(* CoDeSys 2.3 export: geometry.st *)

(* POU Math/Geometry/CIRCLE_A, ST *)
FUNCTION CIRCLE_A : REAL
VAR_INPUT
	R : REAL;
END_VAR


(*
version 1.1	18. oct. 2008
programmer 	hugo
tested by	oscat

this function calculates the area of a circle with radius R

*)
CIRCLE_A := R * R * math.PI;


(* revision history
hm	22. jan. 2007	rev 1.0
	original version

hm	18. oct. 2008	rev 1.1
	using math constants

*)
END_FUNCTION

(* POU Math/Geometry/CIRCLE_C, ST *)
FUNCTION CIRCLE_C : REAL
VAR_INPUT
	R : REAL;
END_VAR


(*
version 1.1	18. oct. 2008
programmer 	hugo
tested by	oscat

this function calculates the circumference of a circle with radius R

*)
CIRCLE_C := R * math.PI2;


(* revision history
hm	22. jan. 2007	rev 1.0
	original version

hm	18. oct. 2008	rev 1.1
	using math constants

*)
END_FUNCTION

(* POU Math/Geometry/CIRCLE_SEG, ST *)
FUNCTION CIRCLE_SEG : REAL
VAR_INPUT
	R : REAL;
	A : REAL;
END_VAR


(*
version 1.1	18. oct. 2008
programmer 	hugo
tested by	oscat

this function calculates the area of a circle segment with radius R and angle A

*)
CIRCLE_SEG := R * R * math.PI * A / 360.0;


(* revision history
hm	22. jan. 2007	rev 1.0
	original version

hm	18. oct. 2008	rev 1.1
	using math constants

*)
END_FUNCTION

(* POU Math/Geometry/CONE_V, ST *)
FUNCTION CONE_V : REAL
VAR_INPUT
	R : REAL;
	H : REAL;
END_VAR


(*
version 1.1	18. oct. 2008
programmer 	hugo
tested by	oscat

this function calculates the volume of a cone with radius R and height H

*)
CONE_V := R * R * math.PI * H / 3.0;


(* revision history
hm	22. jan. 2007	rev 1.0
	original version

hm	18. oct. 2008	rev 1.1
	using math constants

*)
END_FUNCTION

(* POU Math/Geometry/SPHERE_V, ST *)
FUNCTION SPHERE_V : REAL
VAR_INPUT
	R : REAL;
END_VAR


(*
version 1.1	18. oct. 2008
programmer 	hugo
tested by	oscat

this function calculates the volume of a sphere with radius R

*)
SPHERE_V := R * R * R * math.PI4 / 3.0;


(* revision history
hm	22. jan. 2007	rev 1.0
	original version

hm	18. oct. 2008	rev 1.1
	using math constants

*)
END_FUNCTION
